FUNCTION SquareSignal : REAL
VAR_INPUT
	ymin:				REAL; 	//Minimalwert
	ymax:				REAL; 	//Maximalwert
	w:					REAL; 	//Kreisfrequenz
	yoff:				REAL; 	//yoffset
	t : 				REAL;	//Zeit
END_VAR
VAR
	tempTime:			REAL;
	tempVar:			INT;
END_VAR

tempTime := LMOD(lr_Value:=t,lr_Arg:=(2*PI)/w)/((2*PI)/w);

IF(tempTime >= (0.5)) THEN
	SquareSignal := ymax + yoff;
	RETURN;
ELSE
	SquareSignal := ymin + yoff;
	RETURN;
END_IF

END_FUNCTION

(* stored: Version 1.1.0.1, ProductVersion 3.1.4024.13
   POU SquareSignal: Id {385d91cf-5e74-4427-be55-947bb39d8574}, SpecialFunc None *)
